(*******************************************************************************
 * POU Name:    FB_Syntax_ExhaustiveComments
 * Description: Comprehensive test fixture for ALL TwinCAT 3 IEC 61131-3
 *              comment variants (line //, block (* *), nested, inline).
*******************************************************************************)
FUNCTION_BLOCK FB_Syntax_ExhaustiveComments
VAR_INPUT (* Inputs section *)
    /// <summary>Enable command</summary>
    bEnable : BOOL := FALSE; (* Master enable flag *)
    nSetVal : INT  := 100;   // Target value setpoint
    fLimit  : REAL := 99.5;  (* Upper threshold in [degC] *)
END_VAR
VAR_OUTPUT (* Outputs section *)
    /// <summary>Active status</summary>
    bActive     : BOOL;  (* Currently operational *)
    bError      : BOOL;  // Error indicator
    nStatusCode : UDINT; (* Diagnostic code: 16#0000_0000 = OK *)
END_VAR
VAR_IN_OUT (* In-Out variables *)
    stGlobalCtx : ST_Syntax_Mini; (* Shared context structure *)
END_VAR
VAR (* Internal state variables *)
    // --- 1. Control flags ---
    _bInitDone : BOOL := FALSE; (* First-cycle init marker *)
    _nCycleCnt : UDINT;         // Total executed cycles

    // --- 2. State machine ---
    _nStep    : INT := 0; (* Current step index *)
    _nSubStep : INT := 0; // Secondary step

    // --- 3. Arithmetic values ---
    _fAccum     : LREAL := 0.0; (* Filtered accumulator *)
    _fbTonDelay : TON;          (* Failsafe timer *)

    (*
     * Multi-line block comment inside declaration block
     * Explaining temporary calculation buffers
     *)
    _arrScratch : ARRAY[1..4] OF DINT := [
        10, (* buffer 1 *)
        20, (* buffer 2 *)
        30, (* buffer 3 *)
        40  (* buffer 4 *)
    ];
END_VAR
VAR_TEMP (* Temporary cycle-local variables *)
    _nTempLoop  : INT;  // Loop counter
    _bCondition : BOOL; (* Transient flag *)
END_VAR

// =============================================================================
// 1. NESTED BLOCK COMMENTS & DOC COMMENTS
// =============================================================================
(* Outer comment level 1
   (* Nested comment level 2
      (* Deep nested comment level 3: x := 5; IF y THEN z := 1; END_IF; *)
Back TO level 2
*)
Back TO level 1
*)

/// Triple slash documentation comment
// Standard line comment with special chars: <XML attr="val"> & 'quotes' "double"

// =============================================================================
// 2. COMMENTS INSIDE ARITHMETIC & BOOLEAN EXPRESSIONS
// =============================================================================
_fAccum := _fAccum + (* term 1 *) (LREAL#1.5 * (* term 2 *) DINT_TO_LREAL(nSetVal)) - (* term 3 *) (fLimit / (* term 4 *) 2.0);

_bCondition := (bEnable (* check enable *) AND NOT bError (* check error *)) OR_ELSE (* fallback check *) (_nStep = 999 (* emergency *));

// =============================================================================
// 3. COMMENTS IN IF / ELSIF / ELSE CONTROL FLOW
// =============================================================================
IF (* condition check *) _bCondition THEN // branch 1 taken
    // Internal comment
    _nStep := 10; (* move to running step *)
ELSIF (* alternate check *) bError THEN (* branch error *)
    _nStep := 99; // error recovery step
ELSE (* default fallback *)
    _nStep := 0;  (* stay in idle *)
END_IF
(* end of state check *)
;

// =============================================================================
// 4. COMMENTS IN CASE STATEMENT
// =============================================================================
CASE (* evaluate active step *) _nStep OF
    0 (* Step: Idle *):
        // Idle actions
        IF bEnable THEN
            _nStep := 10; // start cycle
        END_IF

    10 (* Step: Running *), 20 (* Step: Processing *):
        // Active processing
        _nCycleCnt := _nCycleCnt + 1; (* increment cycle *)

    99 (* Step: Error *):
        // Error handling
        bError := TRUE;

ELSE (* Step: Unhandled *)
    _nStep := 0; // return to idle
END_CASE
(* end of case evaluation *)
;

// =============================================================================
// 5. COMMENTS IN LOOPS (FOR, WHILE, REPEAT)
// =============================================================================
FOR _nTempLoop := 1 (* start *) TO 4 (* stop *) BY 1 (* step *) DO
    // Array element update
    _arrScratch[_nTempLoop] := _arrScratch[_nTempLoop] + (* offset *) 1;
    IF _arrScratch[_nTempLoop] > 100 THEN
        CONTINUE; // skip rest of loop
    END_IF
END_FOR
(* end of for loop *)
;

WHILE (* guard condition *) (_nSubStep < 5) AND NOT bError DO
    _nSubStep := _nSubStep + 1; // advance sub-step
    IF _nSubStep >= 3 THEN
        EXIT; (* break early *)
    END_IF
END_WHILE
(* end of while loop *)
;

REPEAT
    _nSubStep := _nSubStep - 1; // decrement
UNTIL (* termination condition *) (_nSubStep <= 0)
END_REPEAT
(* end of repeat loop *)
;

// =============================================================================
// 6. COMMENTS IN FB CALLS & FUNCTION CALLS
// =============================================================================
_fbTonDelay(
        IN := (* trigger signal *) (bEnable AND NOT bError), // enable
        PT := (* duration *) T#500MS                        (* 500 ms delay *)
        ); // timer instance call

bActive := _fbTonDelay.Q; // output assignment

(*******************************************************************************
 * Method: M_DiagnosticReport
 * Summary: Generates diagnostic string with nested comments.
 *******************************************************************************)
METHOD M_DiagnosticReport : STRING(255)
VAR_INPUT
    nDetailLevel : INT; (* 0=brief, 1=full *)
END_VAR
VAR
    sReport : STRING(255); // Output accumulator
END_VAR
// Build report string
IF nDetailLevel > 0 THEN
    (* Full detail formatting *)
    sReport := CONCAT((* prefix *) 'Status: ', (* value *) UDINT_TO_STRING(nStatusCode) );
ELSE
    (* Brief formatting *)
    sReport := 'OK';
END_IF

M_DiagnosticReport := sReport; // Return result
END_METHOD

PROPERTY P_IsReady : BOOL
GET
// Getter logic
P_IsReady := _bInitDone AND NOT bError; (* Ready when initialized and no error *)
END_GET
END_PROPERTY

(* stored: Version 1.1.0.1, ProductVersion 3.1.4024.16
   POU FB_Syntax_ExhaustiveComments: Id {03df462c-ae89-4958-ad07-6a10107ee031}, SpecialFunc None
   Method M_DiagnosticReport: Id {308f5f89-647f-483b-8e4f-776ac774973a}
   Property P_IsReady: Id {4eedcc9f-ac19-4331-b01d-b8d46bf172e4}
   Get Get: Id {10c042e0-a486-4aa5-97ca-62f92f37d99a} *)
